FUNCTION_BLOCK FB_WithEmptyVars
VAR_INPUT
    OneInput : REAL;
END_VAR

METHOD DoesSomething : BOOL
END_METHOD

PROPERTY SomeProperty : REAL
GET
END_GET
SET
END_SET
END_PROPERTY

END_FUNCTION_BLOCK

(* stored: Version 1.1.0.1, ProductVersion 3.1.4024.3
   POU FB_WithEmptyVars: Id {106fe56b-b616-4a50-9a9f-10b6fa9ebaf9}, SpecialFunc None
   Method DoesSomething: Id {9b942f00-b876-4ffe-b4c8-ac0a0f43615a}
   Property SomeProperty: Id {ff352683-7d51-441b-a700-2f80c7229c20}
   Get Get: Id {0498394d-8554-4775-8a47-1f6f5f4e3612}
   Set Set: Id {ab0d6451-72bc-4e52-bc8c-978a54b39b98} *)
